Staubli VAL3: Main.pgx

program Main()
  local num l_nKey
begin
  //

  do
    call Refresh()
    l_nKey=getKey()
    bUserRefresh=false
    call MainKey(l_nKey)
    delay(0)
  until bExit
end
